// TIA Portal V16 export
// export: Created 2021-07-12T14:47:13.9777766Z, ExportSetting WithDefaults, DisplayName Totally Integrated Automation Portal, DisplayVersion V16, DisplayName TIA Portal Version Control Interface, DisplayVersion V16, DisplayName TIA Portal Openness, DisplayVersion V16, DisplayName STEP 7 Professional, DisplayVersion V16, DisplayName STEP 7 Safety, DisplayVersion V16, DisplayName WinCC Professional, DisplayVersion V16
ORGANIZATION_BLOCK "SimaHydTO_Main_HMI"   // OB124, LAD, ProgramCycle
TITLE = SimaHydTO_Main_HMI
{ S7_Optimized_Access := 'TRUE' }
FAMILY : SimaHydTO
VERSION : 1.0
// Organization block information: See Organization block network 1
// stored: AutoNumber true, IsIECCheckEnabled false, SetENOAutomatically false
   VAR_INPUT
      Initial_Call : Bool;   // Initial call of this OB
      Remanence : Bool;   // =True, if remanent data are available
   END_VAR
BEGIN

REGION Network 1 (SCL): SimaHydTO - HMI Interface
   //=============================================================================
   //SIEMENS AG
   //(c)Copyright 2016 All Rights Reserved
   //-----------------------------------------------------------------------------
   //Library:       OB of LSimaHydTO_HMI
   //Tested with:   S7-1500 V2.5
   //Engineering:   TIA Portal V15
   //Restrictions:  -
   //Requirements:  S7-1500(T)
   //Functionality: Connection between HMI and PLC program
   //-----------------------------------------------------------------------------
   //Change log table:
   //Version  Date       Expert in charge Changes applied
   //01.00.00 18.07.2019 ArSc             First released version
   //=============================================================================
END_REGION

REGION Network 2: SimaHydTO - HMI Interface: Function calls of HMI functionality
   // Controlling the functionality of SimaHydTO via HMI
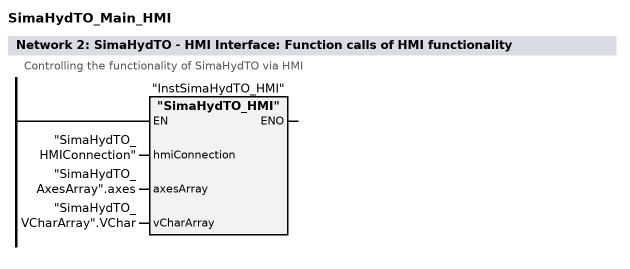
   RUNG wire#powerrail
      "InstSimaHydTO_HMI"(hmiConnection := "SimaHydTO_HMIConnection", axesArray := "SimaHydTO_AxesArray".axes, vCharArray := "SimaHydTO_VCharArray".VChar)
   END_RUNG
   // the same network as SCL:
   "InstSimaHydTO_HMI"(hmiConnection := "SimaHydTO_HMIConnection",   // "SimaHydTO_HMI"
                       axesArray := "SimaHydTO_AxesArray".axes,
                       vCharArray := "SimaHydTO_VCharArray".VChar);
END_REGION
END_ORGANIZATION_BLOCK
